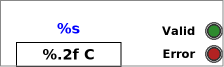
VISUALIZATION TEMPLATE_NOTT_CRYO_TEMPS  // 224x67
VAR_IN_OUT
	m_instance:		FB_CRYO_SENSOR_TEMPERATURE;
END_VAR
    Rectangle (16,16 105x25), "%s", text variable: m_instance.in_sName
    Rectangle (16,42 105x25), "%.2f C", tooltip "Temperature in C", text variable: m_instance.stat.lrTempC
        OnMouseDown: write the text variable via Default
    Group (138,21 86x20)
        Lamp1 (66,0 20x20), variable: m_instance.stat.bValid, style: Lamp-Lamp1-Green
        Rectangle (0,0 60x20), "Valid"
    Group (138,44 86x20)
        Lamp1 (66,0 20x20), variable: m_instance.stat.bError, style: Lamp-Lamp1-Red
        Rectangle (0,0 60x20), "Error"
END_VISUALIZATION

(* stored: Version 1.1.0.1, ProductVersion 3.1.4024.15
   Visu TEMPLATE_NOTT_CRYO_TEMPS: Id {6a15ac34-bf18-499e-a5c7-fc75ed6e8df4} *)
